FUNCTION_BLOCK FB_HMI_EVENTS EXTENDS FB_HMI_COMPONENT
VAR_INPUT
END_VAR
VAR_OUTPUT
END_VAR

END_FUNCTION_BLOCK

(* stored: Version 1.1.0.1, ProductVersion 3.1.4024.14
   POU FB_HMI_EVENTS: Id {e10b79b9-9a23-47ef-a331-5ea43d9a31e2}, SpecialFunc None *)
